Yaskawa INFORM job: VAN-ONDER-NAAR-BOVEN.JBI

/JOB
//NAME VAN-ONDER-NAAR-BOVEN
//POS
///NPOS 5,0,0,0,0,0
///TOOL 1
///POSTYPE PULSE
///PULSE
C00000=9246,34629,-214651,-6202,174139,325719
C00001=9246,-64041,-214651,-6202,174139,325719
C00002=9246,-89754,-52204,-6202,55462,325719
C00003=9246,-89754,67013,-6202,-162538,32377
C00004=-5869,-28950,85500,-7487,-122252,35389
//INST
///DATE 2025/03/05 16:07
///ATTR SC,RW
///GROUP1 RB1
NOP
'==========================================================
' VAN-ONDER-NAAR-BOVEN - Bottom to Top Transition Path
'==========================================================
' Purpose: Moves robot from ONDER (bottom) welding position
'          back to BOVEN (top) welding position safely.
'
' Motion: 5-point joint-interpolated path at full speed (VJ=100)
'         using pulse coordinates. Reverse of VAN-BOVEN-NAAR-ONDER.
'
' Called by: MASTER-START-ML (between ONDER and BOVEN passes)
' Reverse:  VAN-BOVEN-NAAR-ONDER
'==========================================================
' Waypoint 1: Retract from ONDER area
MOVJ C00000 VJ=100.00
' Waypoint 2: Intermediate - begin wrist reorientation
MOVJ C00001 VJ=100.00
' Waypoint 3: Intermediate - wrist flip for BOVEN orientation
MOVJ C00002 VJ=100.00
' Waypoint 4: Intermediate - approach BOVEN side
MOVJ C00003 VJ=100.00
' Waypoint 5: Final BOVEN approach position (same as VAN-BOVEN-NAAR-ONDER start)
MOVJ C00004 VJ=100.00
END
